// TIA Portal V17 export
// export: Created 2025-03-05T08:01:44.8444572Z, ExportSetting WithDefaults, DisplayName Totally Integrated Automation Portal, DisplayVersion V17 Update 8, DisplayName TIA Portal Openness, DisplayVersion V17 Update 8, DisplayName TIA Portal Version Control Interface, DisplayVersion V17, DisplayName SINAMICS Startdrive Advanced, DisplayVersion V17 SP2, DisplayName SINAMICS Startdrive G110M, G120, G120C, G120D, G120P, G115D, DisplayVersion V17 SP2, DisplayName SINAMICS Startdrive G130, G150, S120, S150, SINAMICS MV, S210, DisplayVersion V17 SP2, DisplayName STEP 7 Professional, DisplayVersion V17 Update 8, DisplayName SINUMERIK ONE STEP 7 Toolbox, DisplayVersion V17 Update 12, DisplayName SINUMERIK 840D sl STEP 7 Toolbox, DisplayVersion V17 Update 12, DisplayName STEP 7 Safety, DisplayVersion V17 Update 6, DisplayName WinCC Advanced, DisplayVersion V17 Update 8
DATA_BLOCK "DB7220_MACHINE_OVERVIEW"   // DB7220
{ S7_Optimized_Access := 'FALSE'; DB_Accessible_From_OPC_UA := 'FALSE' }
AUTHOR : ETXETAR
VERSION : 1.0
// stored: AutoNumber false, DBAccessibleFromOPCUA false, DBAccessibleFromWebserver true, IsOnlyStoredInLoadMemory false, IsWriteProtectedInAS false
   VAR RETAIN
      SPINDLES : Struct
         TOOL_IN_SPINDLE_SP11 : Byte;   // NUMBER OF TOOL IN SPINDLE SP11
         TOOL_IN_SPINDLE_SP12 : Byte;   // NUMBER OF TOOL IN SPINDLE SP12
         TOOL_IN_SPINDLE_SP13 : Byte;   // NUMBER OF TOOL IN SPINDLE SP13
         TOOL_IN_SPINDLE_SP14 : Byte;   // NUMBER OF TOOL IN SPINDLE SP14
         TOOL_IN_SPINDLE_SP21 : Byte;   // NUMBER OF TOOL IN SPINDLE SP21
         TOOL_IN_SPINDLE_SP22 : Byte;   // NUMBER OF TOOL IN SPINDLE SP22
         TOOL_IN_SPINDLE_SP23 : Byte;   // NUMBER OF TOOL IN SPINDLE SP23
         TOOL_IN_SPINDLE_SP24 : Byte;   // NUMBER OF TOOL IN SPINDLE SP24
      END_STRUCT;
      EMERGENCY_STOPS : Struct
         STATUS_MPP : Byte;   // MAIN OPERATOR PANEL EMERGENCY STOP 1 STATUS
         STATUS_HT10 : Byte;   // HT8 EMERGENCY STOP 2 STATUS / HT10 EMERGENCY STOP 2 STATUS
         STATUS_LASER_1 : Byte;   // AUXILIARY PANEL EMERGENCY STOP 3 STATUS / LASER UNIT 01 EMERGENCY STOP STATUS
         STATUS_LASER_2 : Byte;   // PART HANDLING DEVICE AUXILIARY PANEL EMERGENCY STOP 4 STATUS / LASER UNIT 02 EMERGENCY STOP STATUS
         STATUS_CHIP_CONV : Byte;   // EMERGENCY STOP 5 STATUS / CHIP CONV PANEL EMERGENCY STOP 5 STATUS
         SPARE : Array[0..9] of Byte;
      END_STRUCT;
      SAFETY_DOORS : Struct
         STATUS_1 : Byte;   // LOAD/UNLOAD SAFETY DOOR 1 STATUS / UNIT 01 MAIN SAFETY DOOR STATUS
         STATUS_2 : Byte;   // MAGAZINE 01R SAFETY DOOR 2 STATUS / UNIT 01 STATION 2 SAFETY DOOR STATUS
         STATUS_3 : Byte;   // MAGAZINE 01L SAFETY DOOR 3 STATUS / UNIT 01 STATION 4 SAFETY DOOR STATUS
         STATUS_4 : Byte;   // MACHINING SAFETY DOOR 4 STATUS / UNIT 01 MAINTENANCE SAFETY DOOR STATUS
         STATUS_5 : Byte;   // MACHINING SAFETY DOOR 4 STATUS / UNIT 01 OERLIKON SAFETY DOOR STATUS
         STATUS_6 : Byte;   // MACHINING SAFETY DOOR 4 STATUS / UNIT 02 MAIN SAFETY DOOR STATUS
         STATUS_7 : Byte;   // PART HANDLING DEVICE SAFETY DOOR 5 STATUS / UNIT 02 STATION 2 SAFETY DOOR STATUS
         STATUS_8 : Byte;   // CHIP CRUSHER SAFETY DOOR 6 STATUS / UNIT 02 STATION 4 SAFETY DOOR STATUS
         STATUS_9 : Byte;   // AUTOMATIC DOOR 7 STATUS / UNIT 02 MAINTENANCE SAFETY DOOR STATUS
         STATUS_10 : Byte;   // UNIT 02 OERLIKON SAFETY DOOR STATUS
         SPARE : Array[0..9] of Byte;
      END_STRUCT;
      MACHINE_UNITS : Struct
         STATUS_UNIT_01 : Byte;   // MACHINE UNIT 1 STATUS (STATION 01R) / MACHINE UNIT 1 STATUS (UNIT 01)
         STATUS_UNIT_02 : Byte;   // MACHINE UNIT 2 STATUS (STATION 01L) / MACHINE UNIT 2 STATUS (UNIT 02)
         STATUS_UNIT_03 : Byte;   // MACHINE UNIT 3 STATUS (PART HANDLING DEVICE) / MACHINE UNIT 3 STATUS (UNIT 03)
         STATUS_FIXT : Byte;   // MACHINE UNIT 4 STATUS / MACHINE UNIT 4 STATUS(FIXTURE)
         STATUS_5 : Byte;   // MACHINE UNIT 5 STATUS
         SPARE : Array[0..4] of Byte;
      END_STRUCT;
      UNIT_MODE : Struct
         STATUS_UNIT_01 : Byte;   // MACHINE UNIT 1 STATUS (STATION 01R) / UNIT 1 MODE STATUS (UNIT 01R)
         STATUS_UNIT_02 : Byte;   // MACHINE UNIT 2 STATUS (STATION 01L) / UNIT 2 MODE STATUS (UNIT 01L)
         STATUS_UNIT_03 : Byte;   // MACHINE UNIT 3 STATUS (PART HANDLING DEVICE) / UNIT 3 MODE STATUS (PART HANDLING DEVICE)
         STATUS_FIXT_1 : Byte;   // MACHINE UNIT 4 STATUS / UNIT 4 MODE STATUS (FIXTURE)
         STATUS_6 : Byte;   // MACHINE UNIT 5 STATUS / UNIT 5 MODE STATUS
         SPARE : Array[0..4] of Byte;
      END_STRUCT;
      UNITS_HOME : Struct
         STATUS_UNIT_01 : Byte;   // MACHINE UNIT 1 STATUS (STATION 01R) / UNIT 1 HOME STATUS (UNIT 01R)
         STATUS_UNIT_02 : Byte;   // MACHINE UNIT 2 STATUS (STATION 01L) / UNIT 2 HOME STATUS (UNIT 01L)
         STATUS_UNIT_03 : Byte;   // MACHINE UNIT 3 STATUS (PART HANDLING DEVICE) / UNIT 3 HOME STATUS (PART HANDLING DEVICE)
         STATUS_FIXT_1 : Byte;   // MACHINE UNIT 4 STATUS / UNIT 4 HOME STATUS (FIXTURE)
         STATUS_6 : Byte;   // MACHINE UNIT 5 STATUS / UNIT 5 HOME STATUS
         SPARE : Array[0..4] of Byte;
      END_STRUCT;
      FIXTURE_1 : Struct
         WORKS_STATUS : Byte;
         IMAG_FIXT_1_CLAMPED : Bool;   // IMAGE FIXTURE 1 CLAMPED
         IMAG_FIXT_1_UNCLAMPED : Bool;   // IMAGE FIXTURE 1 UNCLAMPED
         IMAG_FIXT_1_NOT_CLP_UNCL : Bool;   // IMAGE FIXTURE 1 NOT CLAMPED AND UNCLAMPED
      END_STRUCT;
      FIXTURE_2 : Struct
         WORKS_STATUS : Byte;
         IMAG_FIXT_2_CLAMPED : Bool;   // IMAGE FIXTURE 2 CLAMPED
         IMAG_FIXT_2_UNCLAMPED : Bool;   // IMAGE FIXTURE 2 UNCLAMPED
         IMAG_FIXT_2_NOT_CLP_UNCL : Bool;   // IMAGE FIXTURE 2 NOT CLAMPED AND UNCLAMPED
      END_STRUCT;
      B_AXIS_POSITION : Byte;   // B AXIS POSITION
      E_AXIS_POSITION : Byte;   // E AXIS POSITION
   END_VAR
BEGIN
END_DATA_BLOCK
